{attribute 'qualified_only'}
VAR_GLOBAL
	
	GetLocalSystemTime : FB_LocalSystemTime;
	SystemDateTime : STRING;
	SystemDate : STRING;
	SystemTime : STRING;
	SystemMinutes : STRING;
	SystemSeconds : STRING ; 
END_VAR

(* stored: Version 1.1.0.1, ProductVersion 3.1.4024.12
   GVL GVL: Id {7c02da20-e990-4879-8d70-aaecbb4e4478} *)
